FUNCTION SCALE_UDINT_TO_REAL : REAL
VAR_INPUT
	I : UDINT;
	Range_LL : REAL;
	Range_UL : REAL;
END_VAR
VAR
END_VAR

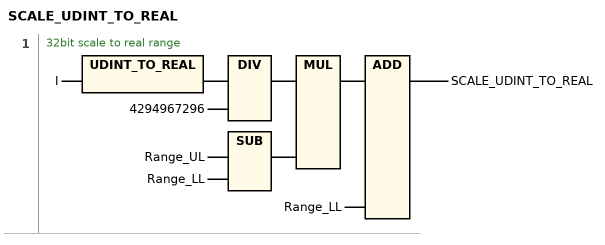
// NETWORK 1
// 32bit scale to real range
SCALE_UDINT_TO_REAL := (UDINT_TO_REAL(I) / 4294967296) * (Range_UL - Range_LL) + Range_LL;

END_FUNCTION

(* stored: Version 1.1.0.1, ProductVersion 3.1.4024.3
   POU SCALE_UDINT_TO_REAL: Id {f2cf4f53-0e96-4639-87d3-c94d63c1e681}, SpecialFunc None *)
